{attribute 'hide_all_locals'}
FUNCTION_BLOCK XtsDisableSequence IMPLEMENTS ITask
VAR_INPUT
END_VAR
VAR_OUTPUT
END_VAR
VAR
	_collisionGroup : REFERENCE TO AXES_GROUP_REF;
	disableGrp : DisableGroup(_collisionGroup);
	removeAllAxes : RemoveAllMoverFromGroup(_collisionGroup);
	grpStop : StopMoverGroup(_collisionGroup);
	State : INT;
	DisableTrigger: BOOL;
	moverNumbers : DINT := 1;
	AllMoversDisabled: BOOL;
	XtsState : REFERENCE TO XtsTrackStates;
	GroupStates : REFERENCE TO CaGroupStates;
	_busy : BOOL;
	_done : BOOL;
	_Error : BOOL;
	i: DINT;
END_VAR
VAR_IN_OUT
	arrMovers : ARRAY[*] OF FB_Mover;
END_VAR

CASE State OF
	0:
		IF DisableTrigger THEN
			DisableTrigger := FALSE;
			XtsState := XtsTrackStates.Disabling;
			_busy := TRUE;
			_done := FALSE;
			_Error := FALSE;
			IF GroupStates.GroupMoving THEN
				grpStop.Execute();
				State := 10;
			ELSE
				State := 20;
				removeAllAxes.RemoveAllMover();
			END_IF
		END_IF
		
	10:
		IF grpStop.Done THEN
			State := 20;
			removeAllAxes.RemoveAllMover();
		END_IF
	
	20:
		IF removeAllAxes.Done THEN
			FOR moverNumbers := LOWER_BOUND(arrMovers,1) TO UPPER_BOUND(arrMovers,1) DO
				arrMovers[moverNumbers].DisableAxis();
			END_FOR
			State := 30;
		END_IF
		
	30:
		AllMoversDisabled := TRUE;
		FOR moverNumbers := LOWER_BOUND(arrMovers,1) TO UPPER_BOUND(arrMovers,1) DO
			AllMoversDisabled := TRUE AND NOT arrMovers[moverNumbers].isEnabled();
		END_FOR
		IF AllMoversDisabled THEN
			State := 50;
			disableGrp.Execute();
		END_IF
		
	50:
		IF disableGrp.Done THEN
			State := 0;
			XtsState := XtsTrackStates.Disabled;
			grpStop.Deceleration := Tc3_Mc3Definitions.MC_DEFAULT;
			grpStop.Jerk := Tc3_Mc3Definitions.MC_DEFAULT;
			_busy := FALSE;
			_done := true;
		END_IF
END_CASE

disableGrp();
removeAllAxes();
grpStop();

{warning 'add method implementation '}
METHOD Abort : BOOL
DisableTrigger := FALSE;
State := 0;
disableGrp.Abort();
removeAllAxes.Abort();
grpStop.Abort();
END_METHOD

{warning 'add property implementation'}
PROPERTY Busy : BOOL
GET
Busy := _busy;
END_GET
END_PROPERTY

METHOD Disable : BOOL
VAR_INPUT
END_VAR
DisableTrigger := true;
END_METHOD

{warning 'add property implementation'}
PROPERTY Done : BOOL
GET
Done := _done;
END_GET
END_PROPERTY

{warning 'add property implementation'}
PROPERTY Error : BOOL
GET
Error := _Error;
END_GET
END_PROPERTY

METHOD FB_init : BOOL
VAR_INPUT
	bInitRetains : BOOL; // if TRUE, the retain variables are initialized (warm start / cold start)
	bInCopyCode : BOOL;  // if TRUE, the instance afterwards gets moved into the copy code (online change)
	collisionGroup : REFERENCE TO AXES_GROUP_REF;
	Status : REFERENCE TO XtsTrackStates;
	GroupState : REFERENCE TO CaGroupStates;
END_VAR
_collisionGroup REF= collisionGroup;
XtsState REF= Status;
GroupStates REF= GroupState;
disableGrp.FB_init(FALSE, FALSE, CAGroup := _collisionGroup);
removeAllAxes.FB_init(FALSE, FALSE, CAGroup := _collisionGroup);
grpStop.FB_init(false,false,CAGroup := _collisionGroup);
END_METHOD

METHOD SetEmergencyDynamics : BOOL
VAR_INPUT
END_VAR
grpStop.Deceleration := Tc3_Mc3Definitions.MC_MAXIMUM;
grpStop.Jerk := Tc3_Mc3Definitions.MC_MAXIMUM;
END_METHOD

END_FUNCTION_BLOCK

(* stored: Version 1.1.0.1, ProductVersion 3.1.4024.6
   POU XtsDisableSequence: Id {ea1d04be-726e-4c7d-baa7-17245f825e22}, SpecialFunc None
   Method Abort: Id {42f8e30f-5183-4033-a58c-7a7275c4a0aa}
   Property Busy: Id {37ba4712-426e-4d01-b6fa-02acf9485af6}
   Get Get: Id {b1cafe39-683e-4a4e-ad04-65ee0fb4226f}
   Method Disable: Id {bc7f7a10-79ff-4b84-9b1c-517283c2b5cf}
   Property Done: Id {eccd7fb2-badb-4f5f-b33a-bdf6f0658780}
   Get Get: Id {a7bff8ff-4014-4380-88b9-a282e05e33b0}
   Property Error: Id {f6b1ac03-fad4-4a5f-9f7c-51705f61776e}
   Get Get: Id {7aba3a07-6d5a-419b-af00-dbecd406527c}
   Method FB_init: Id {e45d29f8-5ba5-4882-9a4e-6018e585a259}
   Method SetEmergencyDynamics: Id {b5418f68-dda4-4664-b66b-f4c1bc501dec} *)
